// Mitsubishi GX Works2 project: math02   PLC: Q02/Q02H

PROGRAM MAIN
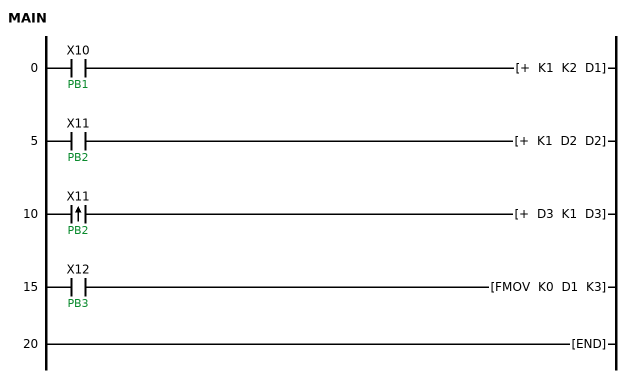
0     LD      X10  ; PB1
      +       K1 K2 D1
5     LD      X11  ; PB2
      +       K1 D2 D2
10    LDP     X11  ; PB2
      +       D3 K1 D3
15    LD      X12  ; PB3
      FMOV    K0 D1 K3
20    END
END_PROGRAM

// device comments not shown above
X0  ; 공급_후
X1  ; 공급_전
X2  ; 드릴_상
X3  ; 드릴_하
X4  ; 송출_후
X5  ; 송출_전
X6  ; 배출_후
X7  ; 배출_전
X8  ; 매거진
X9  ; 비금속
X0A  ; 금속
Y20  ; 공급_전
Y21  ; 공급_후
Y22  ; 드릴_하강
Y23  ; 송출_전
Y24  ; 송출_후
Y25  ; 배출_전
Y26  ; 배출_후
Y27  ; 컨베어
Y28  ; 가공드
Y29  ; 적색
Y2A  ; 황색
Y2B  ; 녹색
